(* PLC project ifmCR711S_TemplateProject, CODESYS CODESYS V3.5 SP11 *)
(* stored: creationDateTime 2026-08-04T14:40:59.4602137, version 2.4.10.0, modificationDateTime 2026-08-04T14:25:20.5601505, organization ifm electronic *)
(* Project template with CR711S configured 2.25MByte Standard 2.25MByte Safety *)

PROGRAM SFC_TEST
  VAR
    SensorA : BOOL;
    SensorB : BOOL;
  END_VAR

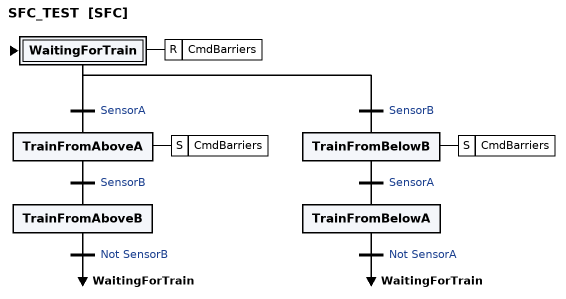
INITIAL_STEP WaitingForTrain:
  CmdBarriers(R);
END_STEP
TRANSITION FROM WaitingForTrain TO TrainFromAboveA
  := SensorA;
END_TRANSITION
TRANSITION FROM WaitingForTrain TO TrainFromBelowB
  := SensorB;
END_TRANSITION
STEP TrainFromAboveA:
  CmdBarriers(S);
END_STEP
TRANSITION FROM TrainFromAboveA TO TrainFromAboveB
  := SensorB;
END_TRANSITION
STEP TrainFromAboveB:
END_STEP
TRANSITION FROM TrainFromAboveB TO WaitingForTrain
  := Not SensorB;
END_TRANSITION
STEP TrainFromBelowB:
  CmdBarriers(S);
END_STEP
TRANSITION FROM TrainFromBelowB TO TrainFromBelowA
  := SensorA;
END_TRANSITION
STEP TrainFromBelowA:
END_STEP
TRANSITION FROM TrainFromBelowA TO WaitingForTrain
  := Not SensorA;
END_TRANSITION
END_PROGRAM
